Universal Robots PolyScope program: Gripper.urp

Program Gripper (createdIn=3.4.0.265 lastSavedIn=3.4.0.265 directory=/programs/usbdisk/GRIPPER installation=Pick_and_Place robotSerialNumber=2016330596)
Calibrated DH parameters: a=[-0.000081, -0.205745, -0.180007, 0.000061, 0.000074, 0]; d=[0.151515, 47.369588, 6.717024, -53.973819, 0.085293, 0.082299]; alpha=[1.572067, -0.002789, -0.00212, 1.569705, -1.570221, 0]; deltaTheta=[0, -0.570859, 0.003648, 0.567188, -0.00001, -0.000013]
BeforeStart
  var_1 := socket_open("192.168.1.20",30000)
  MoveJ speed 60 deg/s, acceleration 80 deg/s^2 (useActiveTCP=false)
    Waypoint Waypoint_1: TCP in base x=216.757 y=79.987 z=180.378 mm, rx=2.9272 ry=-1.0684 rz=0.0286 rad; joints [51.482, -69.779, -91.014, -110.289, 88.318, 1.67] deg; flange x=215.163 y=85.601 z=366.928 mm, rx=2.9272 ry=-1.0684 rz=0.0286 rad
Robot Program (runOnlyOnce=false motionType=MoveJ speed=1.047198 acceleration=1.396263 useActiveTCP=false)
  Loop While (checkContinuously=false) expression=var_1≟ False
    var_1 := socket_open("192.168.1.20",30000)
    Wait Sleep waitTime=0.05
  Script: socket_send_string("ready")
  Wait Sleep waitTime=0.5
  var_2 := socket_read_ascii_float(1)
  Wait Sleep waitTime=0.5
  SuppressedNode
    var_1 := False
  If var_2[1]≟1
    URCap RG2 (RG - On Robot, On Robot ApS) data=depthCompensate = false
      | width = 100
      | name = RG2(100)
      | force = 40
      | payload = 0.0
    Wait Sleep waitTime=0.1
  ElseIf var_2[1]≟0
    URCap RG2 (RG - On Robot, On Robot ApS) data=depthCompensate = false
      | width = 0
      | name = RG2(0)
      | force = 40
      | payload = 0.0
    Wait Sleep waitTime=0.1
